PROGRAM MAIN
VAR
END_VAR

END_PROGRAM

(* stored: Version 1.1.0.1
   POU MAIN: Id {01e2daed-a312-437a-8aa5-c891de0de905} *)
